RoboDK station: PanelRootBottom.rdk

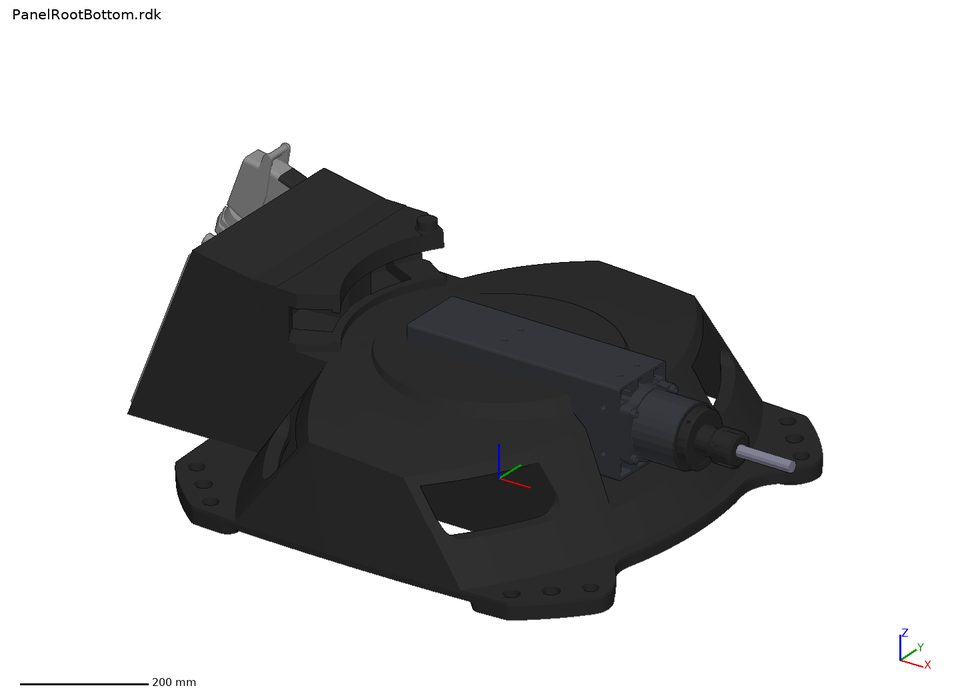
[picture v0: the station drawn from its stored meshes, robots at their saved joint values, targets as dots, program paths as lines]
Station Final (saved by RoboDK 5.2.3). Poses are relative to the parent item; angles as X-Y-Z fixed-axis rotations.
  - frame KUKA KR 210 R2700 extra Base at (0, 0, 0) mm
    - frame Frame_2 at (1500, 1000, 500) mm
    - robot KUKA KR 210 R2700 extra: 6 axes, payload 210 kg, reach 2696 mm, repeatability 0.06 mm, weight 1068 kg
        joint limits [-185, -140, -120, -350, -125, -350] to [185, -5, 155, 350, 125, 350]; home [0, -90, 90, 0, 0, 0]; saved at [-62.962, -88.076, 98.877, 95.463, 63.479, -102.089]
      - tool Spindle, TCP at (557.2, 0, 176) mm, rotated rx 0 ry 90 rz 0 deg, size 692.9 x 170 x 256 mm
  - Python program FinalRobotPlan (listed below)

--- Python program FinalRobotPlan ---
from robolink import *
from robodk import *

data = open('AE1222-2021-GROUP-E09H-CoordinateFile-PanelRootBottom.txt')






# read table and get rid of fat
x = 1000
y = 1000
z = 1000


table = []
test = []

for line in data:
    row = line.split('\t')
    for i in range(7):
        del row[-1]
    res = [float(i) for i in row]
    res[0] += x
    res[1] += y
    res[2] += z
    table.append(res)
print(table)




RDK = Robolink()


RDK.Render(False)


list_items = RDK.ItemList()
for item in list_items:
    if item.Name().startswith('Auto'):
        item.Delete()


robot = RDK.ItemUserPick('Select a robot', ITEM_TYPE_ROBOT)


RDK.Render(True)


if not robot.Valid():
    quit()


reference = robot.Parent()


robot.setPoseFrame(reference)


pose_ref = robot.Pose()
print(Pose_2_TxyzRxyz(pose_ref))




ref = pose_ref
ref.setPos([1000,1000,1500,180,0,180])

robot.MoveJ(ref)

for i in range(len(table)):

    pose_i = pose_ref
    pose_i.setPos(table[i])


    robot.MoveL(pose_i)


ref = pose_ref
ref.setPos([1000,1000,1500,180,0,180])

robot.MoveJ(ref)

quit()
